Staubli VAL3: init.pgx

public program init()
begin
  // Copyright (c) 2021, Institute for Factory Automation and Production Systems (FAPS)
  //
  // Licensed under the Apache License, Version 2.0 (the "License");
  // you may not use this file except in compliance with the License.
  // You may obtain a copy of the License at
  //
  //     http://www.apache.org/licenses/LICENSE-2.0
  //
  // Unless required by applicable law or agreed to in writing, software
  // distributed under the License is distributed on an "AS IS" BASIS,
  // WITHOUT WARRANTIES OR CONDITIONS OF ANY KIND, either express or implied.
  // See the License for the specific language governing permissions and
  // limitations under the License.


  UNKNOWN     = -1
  USER_IN     =  1
  VALVE_OUT   =  2
  BASIC_IN    =  3
  BASIC_OUT   =  4
  BASIC_IN_2  =  5
  BASIC_OUT_2 =  6
end
